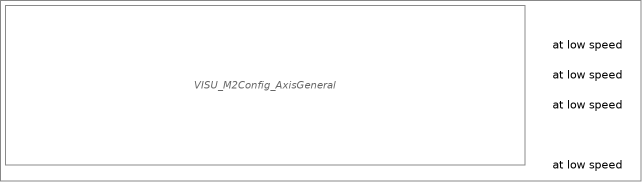
VISUALIZATION VISU_M2Config_ZAxis_General  // 642x182
VAR_IN_OUT
    editable : M2ZAxisConfig;
	active : M2ZAxisConfig;
END_VAR
    Frame (5,5 520x160)
        shows VISU_M2Config_AxisGeneral(editable := editable.general, active := active.general)
    Label (535,30 105x30), "at low speed"
    Label (535,60 105x30), "at low speed"
    Label (535,90 105x30), "at low speed"
    Label (535,150 105x30), "at low speed"
END_VISUALIZATION

(* stored: Version 1.1.0.1, ProductVersion 3.1.4019.2
   Visu VISU_M2Config_ZAxis_General: Id {7b9784da-3540-497a-91d2-b1029d873102} *)
